(* CODESYS project Sejf.project

Project tree, tasks and I/O mapping:
  Device : CODESYS Control Win V3, 3S - Smart Software Solutions GmbH, order no. 305021, version 3.5.8.10
    application Application
      libraries: Standard, * (System)
      task MainTask (cyclic, interval t#20ms, priority 1) calls PLC_PRG
      task VISU_TASK (cyclic, interval 100 ms, priority 31) calls VisuElems.Visu_Prg
      program PLC_PRG [ST]
      visualisation Visualization
  text list GlobalTextList
*)

// Device/Application/PLC_PRG
PROGRAM PLC_PRG
VAR
	GREEN: TON;	
	RED: TON;
	BLOCKED: TON;

	//Deklaracja przycisków
	ONE_B : BOOL;
	TWO_B : BOOL;
	THREE_B : BOOL;
	FOUR_B : BOOL;
	FIVE_B : BOOL;
	SIX_B : BOOL;
	SEVEN_B : BOOL;
	EIGHT_B : BOOL;
	NINE_B : BOOL;
	OK : BOOL;
	
	//Deklaracja wartości przycisków
	ONE : INT := 1;
	TWO : INT := 2;
	THREE : INT := 3;
	FOUR : INT := 4;
	FIVE : INT := 5;
	SIX : INT := 6;
	SEVEN : INT := 7;
	EIGHT : INT := 8;
	NINE : INT := 9;
	
	COUNTER : INT := 1;
	//Kontrolki dostępu
	ACCESS : BOOL := FALSE;
	ACCESS_DENIED : BOOL := FALSE;
	
	//Zmienne do przechowania kombinacji
	MEMORY_1 : INT;
	MEMORY_2 : INT;
	MEMORY_3 : INT;
	MEMORY_4 : INT;
END_VAR

//Wykopnuję program dopóki nie osiągnę trzech błędnych odpowiedzi (licząc od zera)
WHILE COUNTER < 3 DO
	//Ustawiam początkowe wartości 'pamięci', są to wartości spoza zakresu 1-9, aby móc kontrolować dane wejściowe
	MEMORY_1 := -1;
	MEMORY_2 := -1;
	MEMORY_3 := -1;
	MEMORY_4 := -1;
	
	//Ustawiam kontrolę dostępu jako 'BRAK DOSTĘPU'
	ACCESS := FALSE;
	ACCESS_DENIED := FALSE;
	
	
	//Sprawdzam dla każdej kolejnej wartości 'pamięci' jaki został naciśniety klawisz i taką wartość pamiętam w tejże 'pamięci'
	WHILE MEMORY_1 = -1 DO
		IF ONE_B = TRUE THEN
			MEMORY_1 := ONE;
		ELSIF TWO_B = TRUE THEN
			MEMORY_1 := TWO;
		ELSIF THREE_B THEN
			MEMORY_1 := THREE;
		ELSIF FOUR_B THEN
			MEMORY_1 := FOUR;
		ELSIF FIVE_B THEN
			MEMORY_1 := FIVE;
		ELSIF SIX_B THEN
			MEMORY_1 := SIX;
		ELSIF SEVEN_B THEN
			MEMORY_1 := SEVEN;
		ELSIF EIGHT_B THEN
			MEMORY_1 := EIGHT;
		ELSIF NINE_B THEN
			MEMORY_1 := NINE;
		END_IF
	END_WHILE
	
	WHILE MEMORY_2 = MEMORY_1 OR MEMORY_2 = -1 DO
		IF ONE_B = TRUE THEN
			MEMORY_2 := ONE;
		ELSIF TWO_B = TRUE THEN
			MEMORY_2 := TWO;
		ELSIF THREE_B THEN
			MEMORY_2 := THREE;
		ELSIF FOUR_B THEN
			MEMORY_2 := FOUR;
		ELSIF FIVE_B THEN
			MEMORY_2 := FIVE;
		ELSIF SIX_B THEN
			MEMORY_2 := SIX;
		ELSIF SEVEN_B THEN
			MEMORY_2 := SEVEN;
		ELSIF EIGHT_B THEN
			MEMORY_2 := EIGHT;
		ELSIF NINE_B THEN
			MEMORY_2 := NINE;
		END_IF
	END_WHILE
	
	WHILE MEMORY_3 = MEMORY_2 OR MEMORY_3 = -1 DO
		IF ONE_B = TRUE THEN
			MEMORY_3 := ONE;
		ELSIF TWO_B = TRUE THEN
			MEMORY_3 := TWO;
		ELSIF THREE_B THEN
			MEMORY_3 := THREE;
		ELSIF FOUR_B THEN
			MEMORY_3 := FOUR;
		ELSIF FIVE_B THEN
			MEMORY_3 := FIVE;
		ELSIF SIX_B THEN
			MEMORY_3 := SIX;
		ELSIF SEVEN_B THEN
			MEMORY_3 := SEVEN;
		ELSIF EIGHT_B THEN
			MEMORY_3 := EIGHT;
		ELSIF NINE_B THEN
			MEMORY_3 := NINE;
		END_IF
	END_WHILE
	
	WHILE MEMORY_4 = MEMORY_3 OR MEMORY_4 = -1 DO
		IF ONE_B = TRUE THEN
			MEMORY_4 := ONE;
		ELSIF TWO_B = TRUE THEN
			MEMORY_4 := TWO;
		ELSIF THREE_B THEN
			MEMORY_4 := THREE;
		ELSIF FOUR_B THEN
			MEMORY_4 := FOUR;
		ELSIF FIVE_B THEN
			MEMORY_4 := FIVE;
		ELSIF SIX_B THEN
			MEMORY_4 := SIX;
		ELSIF SEVEN_B THEN
			MEMORY_4 := SEVEN;
		ELSIF EIGHT_B THEN
			MEMORY_4 := EIGHT;
		ELSIF NINE_B THEN
			MEMORY_4 := NINE;
		END_IF
	END_WHILE
	
	
	//Jeżeli hasło to 1233 i wciśnięto przycisk OK to dostęp zostaje przyznany licznik błednych odpowiedzi 'COUNTER' zostaje wyzerowany i zaświeca się lampka na 5 sekund
	IF MEMORY_1 = 1 AND MEMORY_2 = 2 AND MEMORY_3 = 3 AND MEMORY_4 = 3 AND OK THEN
		ACCESS := TRUE;
		GREEN(IN:= TRUE, PT:= T#5S);
		
		ACCESS := FALSE;
		COUNTER := 0;
	//Jeżeli licznik błędów osiągnie 3 i więcej to program zaświeca czerwoną kontrolkę na 180 sekund i zeruje tenże licznik
	ELSIF COUNTER >= 3 THEN
		ACCESS_DENIED := TRUE;
		BLOCKED(IN:= TRUE, PT:= T#180S);
		COUNTER := 0;
	//Jeżeli użytkownik się pomyli to zaświeca czerwoną lampkę na 10 sekund i zwiększa licznik błędów o jeden
	ELSE 
		ACCESS_DENIED := TRUE;
		RED(IN:= TRUE, PT:= T#10S);
		COUNTER := COUNTER +1;
	END_IF
END_WHILE

END_PROGRAM

// Device/Application/Visualization
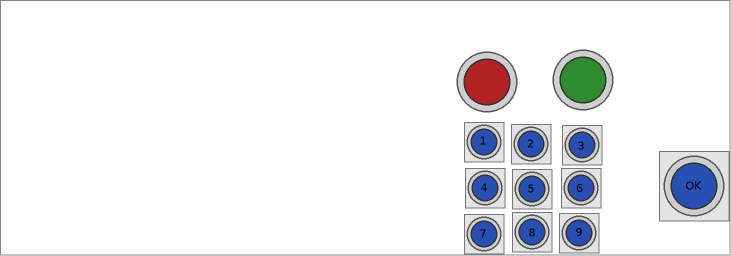
VISUALIZATION Visualization  // 731x256
    Lamp1 (452,47 70x70), variable: PLC_PRG.ACCESS_DENIED, style: Lamp-Lamp1-Red
    Lamp1 (548,45 70x70), variable: PLC_PRG.ACCESS, style: Lamp-Lamp1-Green
    PushSwitch (512,212 40x40), variable: PLC_PRG.EIGHT_B, behaviour: TAP, style: Switch-PushSwitch-Blue
    PushSwitch (464,214 40x40), variable: PLC_PRG.SEVEN_B, behaviour: TAP, style: Switch-PushSwitch-Blue
    PushSwitch (559,213 40x40), variable: PLC_PRG.NINE_B, behaviour: TAP, style: Switch-PushSwitch-Blue
    PushSwitch (465,168 40x40), variable: PLC_PRG.FOUR_B, behaviour: TAP, style: Switch-PushSwitch-Blue
    PushSwitch (512,169 40x40), variable: PLC_PRG.FIVE_B, behaviour: TAP, style: Switch-PushSwitch-Blue
    PushSwitch (561,168 40x40), variable: PLC_PRG.SIX_B, behaviour: TAP, style: Switch-PushSwitch-Blue
    PushSwitch (562,125 40x40), variable: PLC_PRG.THREE_B, behaviour: TAP, style: Switch-PushSwitch-Blue
    PushSwitch (511,124 40x40), variable: PLC_PRG.TWO_B, behaviour: TAP, style: Switch-PushSwitch-Blue
    PushSwitch (464,122 40x40), variable: PLC_PRG.ONE_B, behaviour: TAP, style: Switch-PushSwitch-Blue
    PushSwitch (659,151 70x70), variable: PLC_PRG.OK, behaviour: TAP, style: Switch-PushSwitch-Blue
    Label (473,131 20x20), "1"
    Label (521,132 19x24), "2"
    Label (571,136 20x20), "3"
    Label (474,178 20x20), "4"
    Label (521,178 20x22), "5"
    Label (569,178 21x21), "6"
    Label (473,224 20x20), "7"
    Label (522,223 20x20), "8"
    Label (568,221 22x23), "9"
    Label (677,167 33x38), "OK"
END_VISUALIZATION
